PROGRAM MAIN
VAR
	fbMachine	: FB_Machine;
	bTimeValid	: BOOL;
	bTest		: BOOL;
	bTest2		: BOOL;
END_VAR

fbMachine();
CurrentTime();


//TEst//

METHOD CurrentTime : BOOL
VAR_INPUT
END_VAR
GVL.fbLocalTime(bEnable := TRUE);

IF GVL.fbLocalTime.bValid THEN
	bTimeValid := TRUE;
END_IF

IF bTimeValid THEN
	GVL.iYear 	:= WORD_TO_UINT(GVL.fbLocalTime.systemTime.wYear);
	GVL.iMonth 	:= WORD_TO_UINT(GVL.fbLocalTime.systemTime.wMonth);
	GVL.iDay 	:= WORD_TO_UINT(GVL.fbLocalTime.systemTime.wDay);
	GVL.iHour 	:= WORD_TO_UINT(GVL.fbLocalTime.systemTime.wHour);
	GVL.iMinute := WORD_TO_UINT(GVL.fbLocalTime.systemTime.wMinute);
	GVL.iSecond := WORD_TO_UINT(GVL.fbLocalTime.systemTime.wSecond);
END_IF
END_METHOD

END_PROGRAM

(* stored: Version 1.1.0.1, ProductVersion 3.1.4024.12
   POU MAIN: Id {a5364a73-dda7-4b59-b949-53d76c31a94b}, SpecialFunc None
   Method CurrentTime: Id {2bfafcd3-c480-40dd-83bd-82b250af4621} *)
